Staubli VAL3: start.pgx

program start()
begin
end
